//=============================================================================
// FB_Purge | VERIFIED 8.2.26 DA
//-----------------------------------------------------------------------------
//
// MECHANISM - it is a repeating DRAIN / EQUILIBRATE cycle, not a one-shot:
//   * A pressure band is built around the target setpoint:
//       upper = TSP + band 
//       lower = TSP - band 
//   * Purge only proceeds while upstream pressure is inside that band.
//   * Cycle, gated by "OK to purge" latch:
//       1. Open drain valve SV1 for tDrainOpen 
//       2. Close SV1, wait tEquilibrate to let water settle and for the boiler
//			pressuer loop to raise the upstream pressure to within the range
//       3. If the EMPTY switch (LS3) now reads empty -> purge complete.
//          Otherwise, if still in band, re-open SV1 and repeat.
//   * Overall watchdog: if the cycle runs longer than tPurgeTimeout -> bPurgeFault
//   * After complete: water fill is allowed and the state machine advances
//     to SetDiffPressure
//
// Reports intent only:
//   qDrainValve -> FB_OutputHandler -> GVL_IO.qxSv1Drain (single writer).
//   bPurgeComplete -> FB_StateMachine (S11 -> S13 transition).
//   bPurgeTimeout  -> FB_FaultMonitor (latches the fault, like every other).
//=============================================================================
FUNCTION_BLOCK FB_Purge
VAR_INPUT
    bEnable         		: BOOL;    // TRUE while state = PurgeVessel
    rUpstreamPress  		: REAL;    // upstream pressure [Torr]
    bEmptyFiltered  		: BOOL;    // filtered LS3 empty switch
END_VAR             		
VAR_OUTPUT          		
    qDrainValve     		: BOOL;    // -> FB_OutputHandler -> SV1 drain
    bPurgeComplete  		: BOOL;    // -> state machine
    bPurgeTimeout   		: BOOL;    // -> FaultMonitor Momentary report
    bInPressureBand 		: BOOL;    // diagnostic: pressure within purge band
END_VAR
VAR
    bOkToPurge      		: BOOL;    // "OK to purge" drain-phase latch
    bTimeoutRetryUsed		: BOOL;	   //
	rPressureBandUpper      : REAL;    // 
    rPressureBandLower      : REAL;    // 

    tonDrainOpen    		: TON;     // valve-open dwell
    tonEquilibrate  		: TON;     // valve-closed settle
    tonPurgeTimeout 		: TON;     // overall watchdog
END_VAR

IF NOT bEnable THEN
    qDrainValve       := FALSE;
    bOkToPurge        := FALSE;
    bPurgeComplete    := FALSE;
    bPurgeTimeout     := FALSE;
    bTimeoutRetryUsed := FALSE;
    tonDrainOpen(IN := FALSE);
    tonEquilibrate(IN := FALSE);
    tonPurgeTimeout(IN := FALSE);
    RETURN;
END_IF
// NOTE: the state machine must hold bEnable TRUE for the WHOLE PurgeVessel
// state. Dropping it the moment purge finishes lands here and wipes
// bPurgeComplete, which would restart the blowdown.

//--- pressure band (rung 102) ------------------------------------------------
// Parameters are owned by whoever computes the atmospheric reference. This FB
// only reads them.
rPressureBandUpper := GVL_SysParameters.rPurgeTargetPressure + GVL_SysParameters.rPurgeBand;
rPressureBandLower := GVL_SysParameters.rPurgeTargetPressure - GVL_SysParameters.rPurgeBand;
bInPressureBand    := (rUpstreamPress >= rPressureBandLower)
                  AND (rUpstreamPress <  rPressureBandUpper);

//--- latch the cycle once the boiler reaches the band (rung 105) -------------
// Latch only. The valve stays shut; the first thing that happens is a settle.
IF (NOT bOkToPurge) AND (NOT bPurgeComplete) AND bInPressureBand THEN
    bOkToPurge := TRUE;
END_IF

IF bOkToPurge THEN
    //--- drain-open dwell (rungs 106-107) ------------------------------------
    tonDrainOpen(IN := qDrainValve, PT := GVL_SysParameters.tDrainOpen);
    IF tonDrainOpen.Q THEN
        qDrainValve := FALSE;
    END_IF

    //--- settle dwell, runs whenever the valve is shut (rung 108) ------------
    // Self-rearming: opening the valve drops IN, which resets it.
    tonEquilibrate(IN := NOT qDrainValve, PT := GVL_SysParameters.tEquilibrate);

    //--- end of each settle: done, or blow down again (rungs 109-110) --------
    IF tonEquilibrate.Q THEN
        IF bEmptyFiltered THEN
            bOkToPurge     := FALSE;
            bPurgeComplete := TRUE;
            qDrainValve    := FALSE;
        ELSIF bInPressureBand THEN
            qDrainValve := TRUE;
        END_IF
        // else: pressure fell out of band - hold here until the boiler
        // loop brings it back, then open. (Legacy rung 110 does the same.)
    END_IF

    //--- watchdog, one free retry (rungs 111-113) ----------------------------
    tonPurgeTimeout(IN := TRUE, PT := GVL_SysParameters.tPurgeTimeout);
    IF tonPurgeTimeout.Q THEN
        IF bTimeoutRetryUsed THEN
            bPurgeTimeout := TRUE;
        ELSE
            bTimeoutRetryUsed := TRUE;
            tonPurgeTimeout(IN := FALSE);   // restart for the second window
        END_IF
    END_IF
ELSE
    qDrainValve := FALSE;                   // rung 104
    tonDrainOpen(IN := FALSE);
    tonEquilibrate(IN := FALSE);
    tonPurgeTimeout(IN := FALSE);
    bPurgeTimeout := FALSE;
END_IF

END_FUNCTION_BLOCK

(* stored: Version 1.1.0.1, ProductVersion 3.1.4026.18
   POU FB_Purge: Id {4b1888ad-81a3-443e-843b-d656ed8d9276}, SpecialFunc None *)
